Fanuc KAREL source: wusemaxaccel.kl

PROGRAM wusemaxaccel
%NOLOCKGROUP
VAR
  p : POSITION
  q : POSITION
  i : INTEGER
  r : REAL
BEGIN
  WITH $USEMAXACCEL = TRUE MOVE TO p
END wusemaxaccel
